// TwinCAT 3 PLC project SortationLib
// ProgramVersion: 3.1.4023.0
// libraries:
//   Tc2_Standard, * (Beckhoff Automation GmbH)
//   Tc2_System, * (Beckhoff Automation GmbH)
//   Tc3_Module, * (Beckhoff Automation GmbH)
// project tree:
//   / PlcTask.TcTTO
//   POUs/ MAIN.TcPOU, TONOFF.TcPOU
// real-time tasks:
//   TASK PlcTask: cycle T#10ms, priority 20, ADS port 350

CONFIGURATION SortationLib
    RESOURCE PLC ON TwinCAT3
        TASK PlcTask(INTERVAL := T#10ms, PRIORITY := 20);
        PROGRAM MAIN WITH PlcTask : MAIN;
    END_RESOURCE
END_CONFIGURATION

// ---- POUs/MAIN.TcPOU
PROGRAM MAIN
VAR
END_VAR

END_PROGRAM

// ---- POUs/TONOFF.TcPOU
FUNCTION_BLOCK TONOFF
VAR_INPUT
	IN: BOOL;
	PT:TIME;
END_VAR
VAR_OUTPUT
	Q:BOOL;
END_VAR
VAR
	timeOn:TON;
	timeOff:TOF;
	state: INT;
	Timer: INT;
END_VAR

timeOn(IN:=IN,PT:=PT,Q=>,ET=>);
timeOff(In:=timeOn.Q,PT:=PT,Q=>Q,ET=>);

END_FUNCTION_BLOCK
